// TIA Portal V16 export
// export: Created 2024-09-05T17:39:21.6033356Z, ExportSetting WithDefaults, DisplayName Totally Integrated Automation Portal, DisplayVersion V16 Update 6, DisplayName TIA Portal Version Control Interface, DisplayVersion V16 Update 2, DisplayName TIA Portal Openness, DisplayVersion V16 Update 6, DisplayName STEP 7 Professional, DisplayVersion V16 Update 6, DisplayName STEP 7 Safety, DisplayVersion V16, DisplayName WinCC Advanced, DisplayVersion V16 Update 6
DATA_BLOCK "PartsDataTransfer_DB"   // DB4
VERSION : 0.1
// stored: AutoNumber true, DBAccessibleFromOPCUA true, InstanceOfName PartsDataTransfer, InstanceOfType FB
"PartsDataTransfer"
   // VAR
   //    gripperClose : R_TRIG;
   //    gripperOpen { S7_SetPoint := 'True'} : R_TRIG;
   //    gripperOpenPartial { S7_SetPoint := 'True'} : R_TRIG;
   // END_VAR
BEGIN
   gripperClose.CLK := FALSE;
   gripperClose.Q := FALSE;
   gripperClose.Stat_Bit := FALSE;
   gripperOpen.CLK := TRUE;
   gripperOpen.Q := FALSE;
   gripperOpen.Stat_Bit := TRUE;
   gripperOpenPartial.CLK := TRUE;
   gripperOpenPartial.Q := FALSE;
   gripperOpenPartial.Stat_Bit := TRUE;
END_DATA_BLOCK
